// TIA Portal V17 export
// export: Created 2025-03-07T09:17:50.1684756Z, ExportSetting WithDefaults, DisplayName Totally Integrated Automation Portal, DisplayVersion V17 Update 8, DisplayName TIA Portal Openness, DisplayVersion V17 Update 8, DisplayName TIA Portal Version Control Interface, DisplayVersion V17, DisplayName SINAMICS Startdrive Advanced, DisplayVersion V17 SP2, DisplayName SINAMICS Startdrive G110M, G120, G120C, G120D, G120P, G115D, DisplayVersion V17 SP2, DisplayName SINAMICS Startdrive G130, G150, S120, S150, SINAMICS MV, S210, DisplayVersion V17 SP2, DisplayName STEP 7 Professional, DisplayVersion V17 Update 8, DisplayName SINUMERIK ONE STEP 7 Toolbox, DisplayVersion V17 Update 12, DisplayName SINUMERIK 840D sl STEP 7 Toolbox, DisplayVersion V17 Update 12, DisplayName STEP 7 Safety, DisplayVersion V17 Update 6, DisplayName WinCC Advanced, DisplayVersion V17 Update 8
DATA_BLOCK "DB2109_STATION_3_LIGHT_U01"   // DB2109
{ S7_Optimized_Access := 'FALSE'; DB_Accessible_From_OPC_UA := 'FALSE' }
AUTHOR : ETXETAR
VERSION : 1.0
// stored: AutoNumber false, DBAccessibleFromOPCUA false, DBAccessibleFromWebserver true, IsOnlyStoredInLoadMemory false, IsWriteProtectedInAS false
   VAR RETAIN
      I_CIRCUIT_BREAKER : Bool;   // CIRCUIT BREAKER INPUT
      I_SELECTOR_ON : Bool;   // SELECTOR ON INPUT
      SWITCH_ON_GENERAL_CONDITIONS : Bool;   // SWITCH ON GENERAL CONDITIONS
      SWITCH_ON_INITIAL_CONDITIONS : Bool;   // SWITCH ON INITIAL CONDITIONS
      SWITCH_ON_MANUAL_REQUEST : Bool;   // SWITCH ON MANUAL REQUEST
      SWITCH_ON_AUTO_REQUEST : Bool;   // SWITCH ON AUTO REQUEST
      SWITCH_ON_GLOBAL_REQUEST : Bool;   // SWITCH ON GLOBAL REQUEST
      SWITCH_ON_COMMAND : Bool;   // SWITCH ON COMMAND
      SWITCH_ON : Bool;   // SWITCH ON
      IN_SERVICE : Bool;   // IN SERVICE
      SWITCH_OFF_GENERAL_CONDITIONS : Bool;   // SWITCH OFF GENERAL CONDITIONS
      SWITCH_OFF_INITIAL_CONDITIONS : Bool;   // SWITCH OFF INITIAL CONDITIONS
      SWITCH_OFF_MANUAL_REQUEST : Bool;   // SWITCH OFF MANUAL REQUEST
      SWITCH_OFF_AUTO_REQUEST : Bool;   // SWITCH OFF AUTO REQUEST
      SWITCH_OFF_GLOBAL_REQUEST : Bool;   // SWITCH OFF GLOBAL REQUEST
      SWITCH_OFF_COMMAND : Bool;   // SWITCH OFF COMMAND
      SWITCH_OFF : Bool;   // SWITCH OFF
      OUT_OF_SERVICE : Bool;   // OUT OF SERVICE
      SWITCH_ON_GENERAL_CONDITIONS_HELP : Bool;   // SWITCH ON GENERAL CONDITIONS HELP
      SWITCH_ON_INITIAL_CONDITIONS_HELP : Bool;   // SWITCH ON INITIAL CONDITIONS HELP
      SWITCH_OFF_GENERAL_CONDITIONS_HELP : Bool;   // SWITCH OFF GENERAL CONDITIONS HELP
      SWITCH_OFF_INITIAL_CONDITIONS_HELP : Bool;   // SWITCH OFF INITIAL CONDITIONS HELP
      SWITCH_ON_GLOBAL_REQUEST_AUX1 : Bool;   // SWITCH ON GLOBAL REQUEST ON AUXILIARY 1
      SWITCH_ON_GLOBAL_REQUEST_AUX2 : Bool;   // SWITCH ON GLOBAL REQUEST ON AUXILIARY 2
      SWITCH_ON_GLOBAL_REQUEST_AUX3 : Bool;   // SWITCH ON GLOBAL REQUEST ON AUXILIARY 3
      SWITCH_OFF_AUTO_REQUEST_AUX : Bool;   // INITIAL AUX 4
      SWITCH_OFF_GLOBAL_REQUEST_AUX : Bool;   // INITIAL AUX 5
      TIMER_SWITCH_OFF_1 : TON_TIME;   // SWITCH OFF GLOBAL REQUEST 1 TIMER
      TIMER_SWITCH_OFF_2 : TON_TIME;   // SWITCH OFF GLOBAL REQUEST 2 TIMER
   END_VAR
BEGIN
   TIMER_SWITCH_OFF_1.PT := T#10M;
   TIMER_SWITCH_OFF_2.PT := T#1H;
END_DATA_BLOCK
